// TIA Portal V18 export
DATA_BLOCK "PLC8_910A2_4RTD_AI_Vars"   // DB11021
{ S7_Optimized_Access := 'FALSE' }
VERSION : 0.1
// stored: AutoNumber false, DBAccessibleFromOPCUA true, IsOnlyStoredInLoadMemory false, IsWriteProtectedInAS false
   VAR
      AI1 { S7_SetPoint := 'True'} : "UDT_RTDadv";   // AHU F Темп. зв. теплоносія (1.57)
      AI2 { S7_SetPoint := 'True'} : "UDT_RTDadv";   // AHU F Темп. припл. пов. (1.56)
      AI3 { S7_SetPoint := 'True'} : "UDT_RTDadv";   // AHU F Кімнатна темп. (1.69)
      AI4 { S7_SetPoint := 'True'} : "UDT_RTDadv";   // Резерв
   END_VAR
BEGIN
   AI1.rValue := 26.03;
   AI1.rFilterSet := 0.0;
   AI1.rCalibration := 0.0;
   AI1.rDiv := 100.0;
   AI1.cFuncSystemID := 10;
   AI1.cFuncVar := 4;
   AI1.iReserv := 0;
   AI2.rValue := 3276.7;
   AI2.rFilterSet := 0.0;
   AI2.rCalibration := 0.0;
   AI2.rDiv := 10.0;
   AI2.cFuncSystemID := 16#01;
   AI2.cFuncVar := 16#06;
   AI2.iReserv := 0;
   AI3.rValue := 26.7;
   AI3.rFilterSet := 0.0;
   AI3.rCalibration := 0.0;
   AI3.rDiv := 100.0;
   AI3.cFuncSystemID := 16#01;
   AI3.cFuncVar := 16#04;
   AI3.iReserv := 0;
   AI4.rValue := 22.39;
   AI4.rFilterSet := 0.0;
   AI4.rCalibration := 0.0;
   AI4.rDiv := 100.0;
   AI4.cFuncSystemID := 16#03;
   AI4.cFuncVar := 16#04;
   AI4.iReserv := 0;
END_DATA_BLOCK
